FUNCTION FLOOR2 (* This is a rounding function which returns the biggest possible integer which is less or equal to X. *)
  (* Standard: 61499-1 *)
  (* Version 1.0, 2025-12-21, Franz Höpfinger *)
  PACKAGE OSCAT::Basic::POUs::Mathematical;
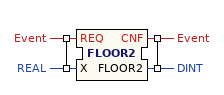
  EVENT_INPUT
    REQ WITH X;
  END_EVENT
  EVENT_OUTPUT
    CNF WITH FLOOR2;
  END_EVENT
  VAR_INPUT
    X : REAL;
  END_VAR
  VAR_OUTPUT
    FLOOR2 : DINT;
  END_VAR
  BODY IN ST:
PACKAGE OSCAT::Basic::POUs::Mathematical;

(* This is a rounding function which returns the biggest possible integer which is less or equal
 * to X. *)
FUNCTION FLOOR2 : DINT
VAR_INPUT
	X : REAL;
END_VAR

(*
 * version 1.1	4. apr. 2008 programmer 	hugo tested by		tobias
 * *
 * This is a rounding function which returns the biggest possible integer which is less or equal to
 * X.
 * floor2(3.14) = 3 floor2(-3.14) = -4
 * *
 *)
FLOOR2 := REAL_TO_DINT(X);
IF DINT_TO_REAL(FLOOR2) > X THEN
	FLOOR2 := FLOOR2 - 1;
END_IF;

END_FUNCTION

(* revision history hm	21. mar. 2008	rev 1.0 originlal version
 * *
 * hm	4. apr. 2008	rev 1.1 added type conversion to avoid warnings under codesys 3.0 *)
  END_BODY
END_FUNCTION
